{attribute 'qualified_only'}
{attribute 'strict'}
TYPE GripperCmd_Enum :
(
	noGrip 	:= 0,
	take	:= 1,
	put		:= 2
);
END_TYPE

(* stored: Version 1.1.0.1, ProductVersion 3.1.4026.13
   DUT GripperCmd_Enum: Id {b80938dc-b405-4653-b69c-ada346329828} *)
